FUNCTION_BLOCK Recipe_10017_DoubleCookiemitTopping
VAR_INPUT
	execute	: BOOL;
	Order	: DUT_RECIPEORDER;
END_VAR
VAR_OUTPUT
	RecipeInfo	: DUT_RECIPEOFFER;
	RecipeDone	: BOOL;	
	InitDone	: BOOL;
END_VAR
VAR
	StepDone	: BOOL;
	Layercnt	: INT := 0;
	OrderLayers	: INT := 1;
END_VAR

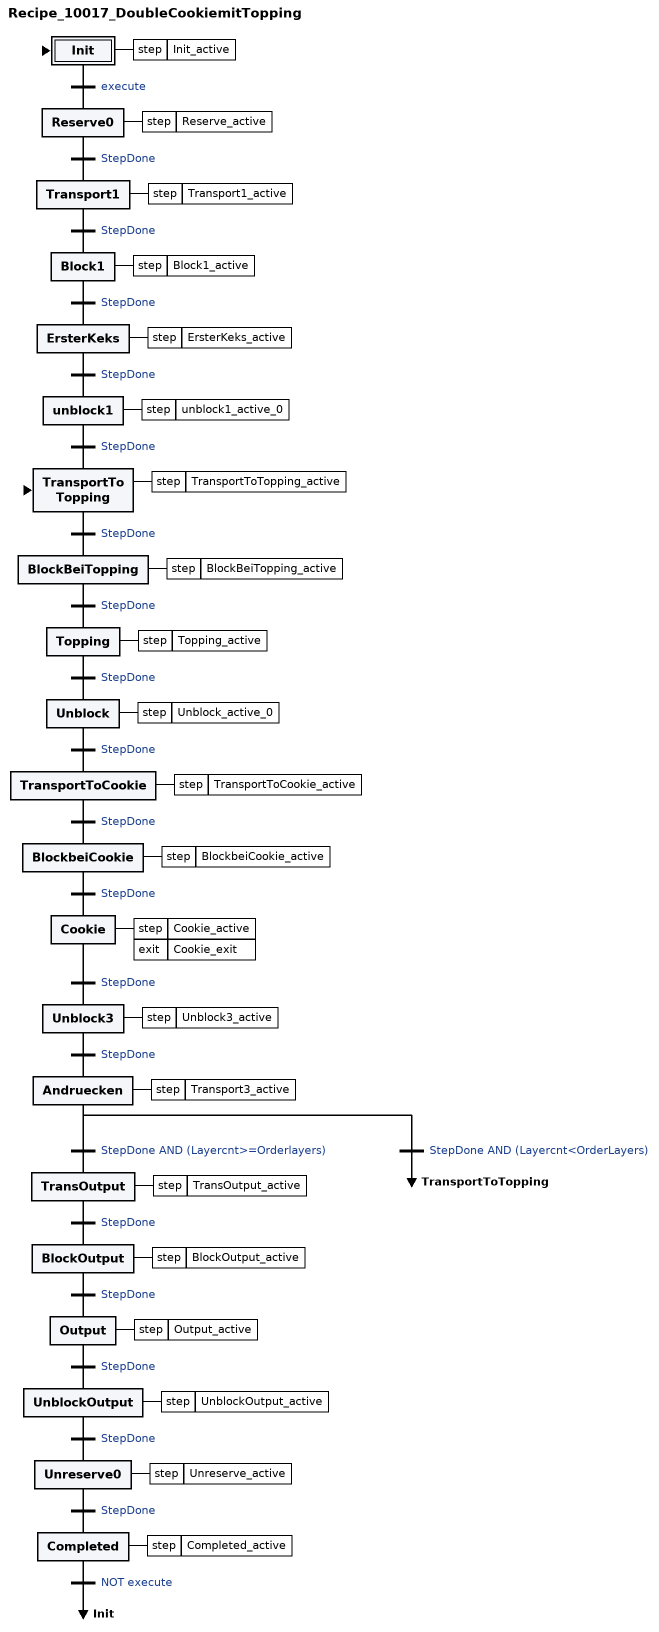
INITIAL_STEP Init:
    Init_active(N);  // step action
END_STEP
TRANSITION FROM Init TO Reserve0
    := execute;
END_TRANSITION
STEP Reserve0:
    Reserve_active(N);  // step action
END_STEP
TRANSITION FROM Reserve0 TO Transport1
    := StepDone;
END_TRANSITION
STEP Transport1:
    Transport1_active(N);  // step action
END_STEP
TRANSITION FROM Transport1 TO Block1
    := StepDone;
END_TRANSITION
STEP Block1:
    Block1_active(N);  // step action
END_STEP
TRANSITION FROM Block1 TO ErsterKeks
    := StepDone;
END_TRANSITION
STEP ErsterKeks:
    ErsterKeks_active(N);  // step action
END_STEP
TRANSITION FROM ErsterKeks TO unblock1
    := StepDone;
END_TRANSITION
STEP unblock1:
    unblock1_active_0(N);  // step action
END_STEP
TRANSITION FROM unblock1 TO TransportToTopping
    := StepDone;
END_TRANSITION
STEP TransportToTopping:
    TransportToTopping_active(N);  // step action
END_STEP
TRANSITION FROM TransportToTopping TO BlockBeiTopping
    := StepDone;
END_TRANSITION
STEP BlockBeiTopping:
    BlockBeiTopping_active(N);  // step action
END_STEP
TRANSITION FROM BlockBeiTopping TO Topping
    := StepDone;
END_TRANSITION
STEP Topping:
    Topping_active(N);  // step action
END_STEP
TRANSITION FROM Topping TO Unblock
    := StepDone;
END_TRANSITION
STEP Unblock:
    Unblock_active_0(N);  // step action
END_STEP
TRANSITION FROM Unblock TO TransportToCookie
    := StepDone;
END_TRANSITION
STEP TransportToCookie:
    TransportToCookie_active(N);  // step action
END_STEP
TRANSITION FROM TransportToCookie TO BlockbeiCookie
    := StepDone;
END_TRANSITION
STEP BlockbeiCookie:
    BlockbeiCookie_active(N);  // step action
END_STEP
TRANSITION FROM BlockbeiCookie TO Cookie
    := StepDone;
END_TRANSITION
STEP Cookie:
    Cookie_active(N);  // step action
    Cookie_exit(P0);  // exit action
END_STEP
TRANSITION FROM Cookie TO Unblock3
    := StepDone;
END_TRANSITION
STEP Unblock3:
    Unblock3_active(N);  // step action
END_STEP
TRANSITION FROM Unblock3 TO Andruecken
    := StepDone;
END_TRANSITION
STEP Andruecken:
    Transport3_active(N);  // step action
END_STEP
TRANSITION FROM Andruecken TO TransOutput
    := StepDone AND (Layercnt>=Orderlayers);
END_TRANSITION
STEP TransOutput:
    TransOutput_active(N);  // step action
END_STEP
TRANSITION FROM TransOutput TO BlockOutput
    := StepDone;
END_TRANSITION
STEP BlockOutput:
    BlockOutput_active(N);  // step action
END_STEP
TRANSITION FROM BlockOutput TO Output
    := StepDone;
END_TRANSITION
STEP Output:
    Output_active(N);  // step action
END_STEP
TRANSITION FROM Output TO UnblockOutput
    := StepDone;
END_TRANSITION
STEP UnblockOutput:
    UnblockOutput_active(N);  // step action
END_STEP
TRANSITION FROM UnblockOutput TO Unreserve0
    := StepDone;
END_TRANSITION
TRANSITION FROM Andruecken TO TransportToTopping
    := StepDone AND (Layercnt<OrderLayers);
END_TRANSITION
STEP Unreserve0:
    Unreserve_active(N);  // step action
END_STEP
TRANSITION FROM Unreserve0 TO Completed
    := StepDone;
END_TRANSITION
STEP Completed:
    Completed_active(N);  // step action
END_STEP
TRANSITION FROM Completed TO Init
    := NOT execute;
END_TRANSITION

ACTION unblock1_active_0:
StepDone := FALSE;

//Skill auswählen
ExecuteSkill.SkillID 		:= 1316;
ExecuteSkill.SkillName	 	:= 'Unblock';

//Parameter setzen

ExecuteSkill.Parameter[1].ID := 1;
ExecuteSkill.Parameter[1].Name := 'TaskID';
ExecuteSkill.Parameter[1].Value := 128 ;


(*
ExecuteSkill.Parameter[2].ID := ;
ExecuteSkill.Parameter[2].Name := '';
ExecuteSkill.Parameter[2].Value := ;
*)

(*
ExecuteSkill.Parameter[3].ID := ;
ExecuteSkill.Parameter[3].Name := '';
ExecuteSkill.Parameter[3].Value := ;
*)

(*
ExecuteSkill.Parameter[4].ID := ;
ExecuteSkill.Parameter[4].Name := '';
ExecuteSkill.Parameter[4].Value := ;
*)

(*
ExecuteSkill.Parameter[5].ID := ;
ExecuteSkill.Parameter[5].Name := '';
ExecuteSkill.Parameter[5].Value := ;
*)



ExecuteSkill();

StepDone := ExecuteSkill.Done;
END_ACTION

ACTION Topping_active:
StepDone := FALSE;

//Skill auswählen
CASE REAL_TO_INT (order.UserParameter[2*LayerCnt].Value) OF
	1: 
		ExecuteSkill.SkillID 		:=  1230;
		ExecuteSkill.SkillName	 	:= 'Strawberry Topping';
	2: 
		ExecuteSkill.SkillID 		:=  1240;
		ExecuteSkill.SkillName	 	:= 'Apple Topping';
	ELSE
		ExecuteSkill.SkillID 		:=  1230;
		ExecuteSkill.SkillName	 	:= 'Strawberry Topping';
END_CASE


//Parameter setzen

ExecuteSkill.Parameter[0].ID := 1;
ExecuteSkill.Parameter[0].Name := 'Amount';
ExecuteSkill.Parameter[0].Value := order.UserParameter[2*LayerCnt + 1].Value ;


(*
ExecuteSkill.Parameter[1].ID := 1;
ExecuteSkill.Parameter[1].Name := 'TaskID';
ExecuteSkill.Parameter[1].Value := 130;
*)
(*
ExecuteSkill.Parameter[2].ID := ;
ExecuteSkill.Parameter[2].Name := '';
ExecuteSkill.Parameter[2].Value := ;
*)

(*
ExecuteSkill.Parameter[3].ID := ;
ExecuteSkill.Parameter[3].Name := '';
ExecuteSkill.Parameter[3].Value := ;
*)

(*
ExecuteSkill.Parameter[4].ID := ;
ExecuteSkill.Parameter[4].Name := '';
ExecuteSkill.Parameter[4].Value := ;
*)

(*
ExecuteSkill.Parameter[5].ID := ;
ExecuteSkill.Parameter[5].Name := '';
ExecuteSkill.Parameter[5].Value := ;
*)

ExecuteSkill();

StepDone := ExecuteSkill.Done;
END_ACTION

ACTION Cookie_active:
StepDone := FALSE;
RecipeDone := FALSE;
//Skill auswählen
ExecuteSkill.SkillID 		:= 1010;
ExecuteSkill.SkillName	 	:= 'Cookie ausgeben';





ExecuteSkill();

StepDone := ExecuteSkill.Done;
END_ACTION

ACTION Transport3_active:
(*StepDone := FALSE;

//Skill auswählen
ExecuteSkill.SkillID 		:= 1320;
ExecuteSkill.SkillName	 	:= 'Transport';

//Parameter setzen

ExecuteSkill.Parameter[3].ID := 3;
ExecuteSkill.Parameter[3].Name := 'Velocity';
ExecuteSkill.Parameter[3].Value := 2800;



ExecuteSkill.Parameter[1].ID :=  1;
ExecuteSkill.Parameter[1].Name := 'TargetPosition X';
ExecuteSkill.Parameter[1].Value := 30 ;
ExecuteSkill.Parameter[1].StringValue := '#DP#-2#XPosition';



ExecuteSkill.Parameter[2].ID := 2;
ExecuteSkill.Parameter[2].Name := 'TargetPosition Z';
ExecuteSkill.Parameter[2].Value := 105;// ZCookieModule - ZCookieModuleCalibration - 2* Cookiethickness + toppingthickness+ Preasureheight  ;



ExecuteSkill.Parameter[4].ID := 4;
ExecuteSkill.Parameter[4].Name := 'Acceleration';
ExecuteSkill.Parameter[4].Value := 2000 ;


(*
ExecuteSkill.Parameter[5].ID := ;
ExecuteSkill.Parameter[5].Name := '';
ExecuteSkill.Parameter[5].Value := ;
*)



ExecuteSkill();

StepDone := ExecuteSkill.Done;
*)
StepDone := TRUE;
END_ACTION

ACTION Completed_active:
RecipeDone := TRUE;
StepDone := FALSE;
Layercnt := 0;
END_ACTION

ACTION BlockbeiCookie_active:
StepDone := FALSE;

//Skill auswählen
ExecuteSkill.SkillID 		:= 1315;
ExecuteSkill.SkillName	 	:= 'Block';

//Parameter setzen

ExecuteSkill.Parameter[1].ID := 1;
ExecuteSkill.Parameter[1].Name := 'TaskID';
ExecuteSkill.Parameter[1].Value := 130;


(*
ExecuteSkill.Parameter[2].ID := ;
ExecuteSkill.Parameter[2].Name := '';
ExecuteSkill.Parameter[2].Value := ;
*)

(*
ExecuteSkill.Parameter[3].ID := ;
ExecuteSkill.Parameter[3].Name := '';
ExecuteSkill.Parameter[3].Value := ;
*)

(*
ExecuteSkill.Parameter[4].ID := ;
ExecuteSkill.Parameter[4].Name := '';
ExecuteSkill.Parameter[4].Value := ;
*)

(*
ExecuteSkill.Parameter[5].ID := ;
ExecuteSkill.Parameter[5].Name := '';
ExecuteSkill.Parameter[5].Value := ;
*)



ExecuteSkill();

StepDone := ExecuteSkill.Done;
END_ACTION

ACTION BlockBeiTopping_active:
StepDone := FALSE;

//Skill auswählen
ExecuteSkill.SkillID 		:= 1315;
ExecuteSkill.SkillName	 	:= 'Block';

//Parameter setzen

ExecuteSkill.Parameter[1].ID := 1;
ExecuteSkill.Parameter[1].Name := 'TaskID';
ExecuteSkill.Parameter[1].Value := 130;


(*
ExecuteSkill.Parameter[2].ID := ;
ExecuteSkill.Parameter[2].Name := '';
ExecuteSkill.Parameter[2].Value := ;
*)

(*
ExecuteSkill.Parameter[3].ID := ;
ExecuteSkill.Parameter[3].Name := '';
ExecuteSkill.Parameter[3].Value := ;
*)

(*
ExecuteSkill.Parameter[4].ID := ;
ExecuteSkill.Parameter[4].Name := '';
ExecuteSkill.Parameter[4].Value := ;
*)

(*
ExecuteSkill.Parameter[5].ID := ;
ExecuteSkill.Parameter[5].Name := '';
ExecuteSkill.Parameter[5].Value := ;
*)



ExecuteSkill();

StepDone := ExecuteSkill.Done;
END_ACTION

ACTION ErsterKeks_active:
StepDone := FALSE;
RecipeDone := FALSE;
//Skill auswählen
ExecuteSkill.SkillID 		:= 1010;
ExecuteSkill.SkillName	 	:= 'Seperate Cookie';


ExecuteSkill();

StepDone := ExecuteSkill.Done;
END_ACTION

ACTION Transport1_active:
StepDone := FALSE;

//Skill auswählen
ExecuteSkill.SkillID 		:= 1320;
ExecuteSkill.SkillName	 	:= 'Transport';

//Parameter setzen

ExecuteSkill.Parameter[3].ID := 3;
ExecuteSkill.Parameter[3].Name := 'Velocity';
ExecuteSkill.Parameter[3].Value := 1500;



ExecuteSkill.Parameter[4].ID := 4 ;
ExecuteSkill.Parameter[4].Name := 'Acceleration';
ExecuteSkill.Parameter[4].Value := 1000 ;



ExecuteSkill.Parameter[1].ID := 1;
ExecuteSkill.Parameter[1].Name := 'TargetPosition X';
ExecuteSkill.Parameter[1].Value := 3200 ;
ExecuteSkill.Parameter[1].StringValue := '#DP#2#XPosition' ;




ExecuteSkill.Parameter[2].ID := 2;
ExecuteSkill.Parameter[2].Name := 'TargetPosition Z';
ExecuteSkill.Parameter[2].Value := ZCookieModule + ZCocktailModuleCalibration;


(*
ExecuteSkill.Parameter[5].ID := ;
ExecuteSkill.Parameter[5].Name := '';
ExecuteSkill.Parameter[5].Value := ;
*)



ExecuteSkill();

StepDone := ExecuteSkill.Done;
END_ACTION

ACTION Production0_active:
StepDone := FALSE;
RecipeDone := FALSE; 
//simulation ausgewählt?
CASE LREAL_TO_INT (order.UserParameter[2].Value) OF

1:
ExecuteSkill.SkillID 		:= 1337;
ExecuteSkill.SkillName	 	:= 'Testskill';

ExecuteSkill();

StepDone := ExecuteSkill.Done;
ELSE StepDone := TRUE;

END_CASE
END_ACTION

ACTION TransportToTopping_active:
StepDone := FALSE;

//Skill auswählen
ExecuteSkill.SkillID 		:= 1320;
ExecuteSkill.SkillName	 	:= 'Transport';

//Parameter setzen

ExecuteSkill.Parameter[3].ID := 3;
ExecuteSkill.Parameter[3].Name := 'Velocity';
ExecuteSkill.Parameter[3].Value := 1000;



ExecuteSkill.Parameter[1].ID :=  1;
ExecuteSkill.Parameter[1].Name := 'TargetPosition X';
ExecuteSkill.Parameter[1].Value := 30 ;
ExecuteSkill.Parameter[1].StringValue := '#DP#2#XPosition';



ExecuteSkill.Parameter[2].ID := 2;
ExecuteSkill.Parameter[2].Name := 'TargetPosition Z';
ExecuteSkill.Parameter[2].Value := ZCremeModule + ZCremeModuleCalibration - Layercnt * ( cookiethickness + toppingthickness);

ExecuteSkill();

StepDone := ExecuteSkill.Done;
END_ACTION

ACTION UnblockOutput_active:
StepDone := FALSE;

//Skill auswählen
ExecuteSkill.SkillID 		:= 1316;
ExecuteSkill.SkillName	 	:= 'Unblock';

//Parameter setzen



(*
ExecuteSkill.Parameter[2].ID := ;
ExecuteSkill.Parameter[2].Name := '';
ExecuteSkill.Parameter[2].Value := ;
*)

(*
ExecuteSkill.Parameter[3].ID := ;
ExecuteSkill.Parameter[3].Name := '';
ExecuteSkill.Parameter[3].Value := ;
*)

(*
ExecuteSkill.Parameter[4].ID := ;
ExecuteSkill.Parameter[4].Name := '';
ExecuteSkill.Parameter[4].Value := ;
*)

(*
ExecuteSkill.Parameter[5].ID := ;
ExecuteSkill.Parameter[5].Name := '';
ExecuteSkill.Parameter[5].Value := ;
*)



ExecuteSkill();

StepDone := ExecuteSkill.Done;
END_ACTION

ACTION BlockOutput_active:
StepDone := FALSE;

//Skill auswählen



ExecuteSkill.SkillID 		:= 1315;
ExecuteSkill.SkillName	 	:= 'Block';

ExecuteSkill();

StepDone := ExecuteSkill.Done;
END_ACTION

ACTION Transport_active:
StepDone := FALSE;

//Skill auswählen

CASE LREAL_TO_INT (order.UserParameter[2].Value) OF

1:
//Skill auswählen
ExecuteSkill.SkillID 		:= 1320;
ExecuteSkill.SkillName	 	:= 'Transport';

//Parameter setzen

ExecuteSkill.Parameter[3].ID :=3 ;
ExecuteSkill.Parameter[3].Name := 'Velocity';
ExecuteSkill.Parameter[3].Value := 1500;



ExecuteSkill.Parameter[1].ID :=1 ;
ExecuteSkill.Parameter[1].Name := 'TargetPosition X';
ExecuteSkill.Parameter[1].StringValue := '#DP#2#XPosition';
ExecuteSkill.Parameter[1].Value := 200 ;


ExecuteSkill.Parameter[2].ID := 2 ;
ExecuteSkill.Parameter[2].Name := 'TargetPosition Z';
ExecuteSkill.Parameter[2].Value := 90 ;



ExecuteSkill.Parameter[4].ID := 4 ;
ExecuteSkill.Parameter[4].Name := 'Acceleration';
ExecuteSkill.Parameter[4].Value := 4500;


(*
ExecuteSkill.Parameter[5].ID := ;
ExecuteSkill.Parameter[5].Name := '';
ExecuteSkill.Parameter[5].Value := ;
*)



ExecuteSkill();

StepDone := ExecuteSkill.Done;
ELSE StepDone := TRUE;

END_CASE
END_ACTION

ACTION Unblock_active:
StepDone := FALSE;

//Skill auswählen
ExecuteSkill.SkillID 		:= 1316;
ExecuteSkill.SkillName	 	:= 'Unblock';

//Parameter setzen

ExecuteSkill.Parameter[1].ID := 1;
ExecuteSkill.Parameter[1].Name := 'TaskID';
ExecuteSkill.Parameter[1].Value := 125;


(*
ExecuteSkill.Parameter[2].ID := ;
ExecuteSkill.Parameter[2].Name := '';
ExecuteSkill.Parameter[2].Value := ;
*)

(*
ExecuteSkill.Parameter[3].ID := ;
ExecuteSkill.Parameter[3].Name := '';
ExecuteSkill.Parameter[3].Value := ;
*)

(*
ExecuteSkill.Parameter[4].ID := ;
ExecuteSkill.Parameter[4].Name := '';
ExecuteSkill.Parameter[4].Value := ;
*)

(*
ExecuteSkill.Parameter[5].ID := ;
ExecuteSkill.Parameter[5].Name := '';
ExecuteSkill.Parameter[5].Value := ;
*)



ExecuteSkill();

StepDone := ExecuteSkill.Done;
END_ACTION

ACTION Production2_active:
StepDone := FALSE;
RecipeDone := FALSE;
//Skill auswählen
ExecuteSkill.SkillID 		:= 1339;
ExecuteSkill.SkillName	 	:= 'ParameterTESTSKILL1339';


ExecuteSkill.Parameter[0].ID := 10;
ExecuteSkill.Parameter[0].Name := 'Blinkfrequenz';
ExecuteSkill.Parameter[0].Value := Order.UserParameter[0].Value*2;


ExecuteSkill();

StepDone := ExecuteSkill.Done;
END_ACTION

ACTION Unblock3_active:
StepDone := FALSE;

//Skill auswählen
ExecuteSkill.SkillID 		:= 1316;
ExecuteSkill.SkillName	 	:= 'Unblock';

//Parameter setzen

ExecuteSkill.Parameter[1].ID := 1;
ExecuteSkill.Parameter[1].Name := 'TaskID';
ExecuteSkill.Parameter[1].Value := 131;


(*
ExecuteSkill.Parameter[2].ID := ;
ExecuteSkill.Parameter[2].Name := '';
ExecuteSkill.Parameter[2].Value := ;
*)

(*
ExecuteSkill.Parameter[3].ID := ;
ExecuteSkill.Parameter[3].Name := '';
ExecuteSkill.Parameter[3].Value := ;
*)

(*
ExecuteSkill.Parameter[4].ID := ;
ExecuteSkill.Parameter[4].Name := '';
ExecuteSkill.Parameter[4].Value := ;
*)

(*
ExecuteSkill.Parameter[5].ID := ;
ExecuteSkill.Parameter[5].Name := '';
ExecuteSkill.Parameter[5].Value := ;
*)



ExecuteSkill();

StepDone := ExecuteSkill.Done;
END_ACTION

ACTION ST40_TransOutput_active:
//RT: 2014.11.23: Mover zum Output
StepDone := FALSE;

//Skill auswählen
ExecuteSkill.SkillID 		:= 1320;
ExecuteSkill.SkillName	 	:= 'Transport';

//Parameter setzen

ExecuteSkill.Parameter[3].ID := 3;
ExecuteSkill.Parameter[3].Name := 'Velocity';
ExecuteSkill.Parameter[3].Value := 300;



ExecuteSkill.Parameter[1].ID :=  1;
ExecuteSkill.Parameter[1].Name := 'TargetPosition X';
ExecuteSkill.Parameter[1].Value := 30 ;
ExecuteSkill.Parameter[1].StringValue := '#DP#2#XPosition';



ExecuteSkill.Parameter[2].ID := 2;
ExecuteSkill.Parameter[2].Name := 'TargetPosition Z';
ExecuteSkill.Parameter[2].Value := ZInputOutput;// ZCookieModule - ZCookieModuleCalibration - 2* Cookiethickness + toppingthickness+ Preasureheight  ;



(* ExecuteSkill.Parameter[4].ID := 4;
ExecuteSkill.Parameter[4].Name := 'Acceleration';
ExecuteSkill.Parameter[4].Value :=0 ;

*)
(*
ExecuteSkill.Parameter[5].ID := ;
ExecuteSkill.Parameter[5].Name := '';
ExecuteSkill.Parameter[5].Value := ;
*)



ExecuteSkill();

StepDone := ExecuteSkill.Done;
END_ACTION

ACTION Block2_active:
StepDone := FALSE;

//Skill auswählen
ExecuteSkill.SkillID 		:= 1315;
ExecuteSkill.SkillName	 	:= 'Block';

//Parameter setzen

ExecuteSkill.Parameter[1].ID := 1;
ExecuteSkill.Parameter[1].Name := 'TaskID';
ExecuteSkill.Parameter[1].Value := 130;


(*
ExecuteSkill.Parameter[2].ID := ;
ExecuteSkill.Parameter[2].Name := '';
ExecuteSkill.Parameter[2].Value := ;
*)

(*
ExecuteSkill.Parameter[3].ID := ;
ExecuteSkill.Parameter[3].Name := '';
ExecuteSkill.Parameter[3].Value := ;
*)

(*
ExecuteSkill.Parameter[4].ID := ;
ExecuteSkill.Parameter[4].Name := '';
ExecuteSkill.Parameter[4].Value := ;
*)

(*
ExecuteSkill.Parameter[5].ID := ;
ExecuteSkill.Parameter[5].Name := '';
ExecuteSkill.Parameter[5].Value := ;
*)



ExecuteSkill();

StepDone := ExecuteSkill.Done;
END_ACTION

ACTION Unblock2_active:
StepDone := FALSE;

//Skill auswählen
ExecuteSkill.SkillID 		:= 1316;
ExecuteSkill.SkillName	 	:= 'Unblock';

//Parameter setzen

ExecuteSkill.Parameter[1].ID := 1;
ExecuteSkill.Parameter[1].Name := 'TaskID';
ExecuteSkill.Parameter[1].Value := 131;


(*
ExecuteSkill.Parameter[2].ID := ;
ExecuteSkill.Parameter[2].Name := '';
ExecuteSkill.Parameter[2].Value := ;
*)

(*
ExecuteSkill.Parameter[3].ID := ;
ExecuteSkill.Parameter[3].Name := '';
ExecuteSkill.Parameter[3].Value := ;
*)

(*
ExecuteSkill.Parameter[4].ID := ;
ExecuteSkill.Parameter[4].Name := '';
ExecuteSkill.Parameter[4].Value := ;
*)

(*
ExecuteSkill.Parameter[5].ID := ;
ExecuteSkill.Parameter[5].Name := '';
ExecuteSkill.Parameter[5].Value := ;
*)



ExecuteSkill();

StepDone := ExecuteSkill.Done;
END_ACTION

ACTION TransOutput_active:
StepDone := FALSE;

//Skill auswählen
ExecuteSkill.SkillID 		:= 1320;
ExecuteSkill.SkillName	 	:= 'Transport';

//Parameter setzen

ExecuteSkill.Parameter[3].ID := 3;
ExecuteSkill.Parameter[3].Name := 'Velocity';
ExecuteSkill.Parameter[3].Value := 280;



ExecuteSkill.Parameter[1].ID :=  1;
ExecuteSkill.Parameter[1].Name := 'TargetPosition X';
ExecuteSkill.Parameter[1].Value := 30 ;
ExecuteSkill.Parameter[1].StringValue := '#DP#2#XPosition';



ExecuteSkill.Parameter[2].ID := 2;
ExecuteSkill.Parameter[2].Name := 'TargetPosition Z';
ExecuteSkill.Parameter[2].Value := ZInputOutput;// ZCookieModule - ZCookieModuleCalibration - 2* Cookiethickness + toppingthickness+ Preasureheight  ;



(* ExecuteSkill.Parameter[4].ID := 4;
ExecuteSkill.Parameter[4].Name := 'Acceleration';
ExecuteSkill.Parameter[4].Value :=0 ;

*)
(*
ExecuteSkill.Parameter[5].ID := ;
ExecuteSkill.Parameter[5].Name := '';
ExecuteSkill.Parameter[5].Value := ;
*)



ExecuteSkill();

StepDone := ExecuteSkill.Done;
END_ACTION

ACTION Cookie_exit:
Layercnt := Layercnt +1;
END_ACTION

ACTION Unblock1_active:
StepDone := FALSE;

//Skill auswählen

CASE LREAL_TO_INT (order.UserParameter[2].Value) OF

1:
ExecuteSkill.SkillID 		:= 1316;
ExecuteSkill.SkillName	 	:= 'Unblock';

ExecuteSkill();

StepDone := ExecuteSkill.Done;
ELSE StepDone := TRUE;

END_CASE
END_ACTION

ACTION Output_active:
StepDone := FALSE;

//Skill auswählen
ExecuteSkill.SkillID 		:= 1403;
ExecuteSkill.SkillName	 	:= 'Output';

//Parameter setzen

ExecuteSkill.Parameter[1].ID := 1;
ExecuteSkill.Parameter[1].Name := 'TaskID';
ExecuteSkill.Parameter[1].Value := Order.TaskID;


(*
ExecuteSkill.Parameter[2].ID := ;
ExecuteSkill.Parameter[2].Name := '';
ExecuteSkill.Parameter[2].Value := ;
*)

(*
ExecuteSkill.Parameter[3].ID := ;
ExecuteSkill.Parameter[3].Name := '';
ExecuteSkill.Parameter[3].Value := ;
*)

(*
ExecuteSkill.Parameter[4].ID := ;
ExecuteSkill.Parameter[4].Name := '';
ExecuteSkill.Parameter[4].Value := ;
*)

(*
ExecuteSkill.Parameter[5].ID := ;
ExecuteSkill.Parameter[5].Name := '';
ExecuteSkill.Parameter[5].Value := ;
*)



ExecuteSkill();

StepDone := ExecuteSkill.Done;
END_ACTION

ACTION Block1_active:
StepDone := FALSE;

//Skill auswählen
ExecuteSkill.SkillID 		:= 1315;
ExecuteSkill.SkillName	 	:= 'Block';

//Parameter setzen

ExecuteSkill.Parameter[1].ID := 1;
ExecuteSkill.Parameter[1].Name := 'TaskID';
ExecuteSkill.Parameter[1].Value := 127;


(*
ExecuteSkill.Parameter[2].ID := ;
ExecuteSkill.Parameter[2].Name := '';
ExecuteSkill.Parameter[2].Value := ;
*)

(*
ExecuteSkill.Parameter[3].ID := ;
ExecuteSkill.Parameter[3].Name := '';
ExecuteSkill.Parameter[3].Value := ;
*)

(*
ExecuteSkill.Parameter[4].ID := ;
ExecuteSkill.Parameter[4].Name := '';
ExecuteSkill.Parameter[4].Value := ;
*)

(*
ExecuteSkill.Parameter[5].ID := ;
ExecuteSkill.Parameter[5].Name := '';
ExecuteSkill.Parameter[5].Value := ;
*)



ExecuteSkill();

StepDone := ExecuteSkill.Done;
END_ACTION

ACTION Block0_active:
StepDone := FALSE;

//Skill auswählen

CASE LREAL_TO_INT (order.UserParameter[2].Value) OF

1:
ExecuteSkill.SkillID 		:= 1315;
ExecuteSkill.SkillName	 	:= 'Block';

ExecuteSkill();

StepDone := ExecuteSkill.Done;
ELSE StepDone := TRUE;

END_CASE
END_ACTION

ACTION Unreserve_active:
StepDone := FALSE;

//Skill auswählen
ExecuteSkill.SkillID 		:= 1311;
ExecuteSkill.SkillName	 	:= 'Unreserve';

//Parameter setzen

ExecuteSkill.Parameter[1].ID := 1;
ExecuteSkill.Parameter[1].Name := 'TaskID';
ExecuteSkill.Parameter[1].Value := 131;


(*
ExecuteSkill.Parameter[2].ID := ;
ExecuteSkill.Parameter[2].Name := '';
ExecuteSkill.Parameter[2].Value := ;
*)

(*
ExecuteSkill.Parameter[3].ID := ;
ExecuteSkill.Parameter[3].Name := '';
ExecuteSkill.Parameter[3].Value := ;
*)

(*
ExecuteSkill.Parameter[4].ID := ;
ExecuteSkill.Parameter[4].Name := '';
ExecuteSkill.Parameter[4].Value := ;
*)

(*
ExecuteSkill.Parameter[5].ID := ;
ExecuteSkill.Parameter[5].Name := '';
ExecuteSkill.Parameter[5].Value := ;
*)



ExecuteSkill();

StepDone := ExecuteSkill.Done;
END_ACTION

ACTION Init_active:
RecipeDone := FALSE;

// Initialisation of Recipe Parameters an name etc
RecipeInfo.Name := 'Double Cookie';
RecipeInfo.Description := 'Butter Cookies framing your choosen Topping';
RecipeInfo.Dummy := FALSE;
RecipeInfo.RecipeID := 10017;	// 
Initdone := TRUE;


//Parameter 0:

	RecipeInfo.UserParameter[0].Dummy 		:= FALSE;
	RecipeInfo.UserParameter[0].Default		:= 1;
	RecipeInfo.UserParameter[0].Description	:= 'Choose your first Topping (Top Layer)';
	RecipeInfo.UserParameter[0].MaxValue	:= 2;
	RecipeInfo.UserParameter[0].MinValue	:= 1;
	RecipeInfo.UserParameter[0].Name		:= 'Topping';
	RecipeInfo.UserParameter[0].Unit		:= 'Strawberry, Apple';
	RecipeInfo.UserParameter[0].Step		:= 1;

//Parameter 1:

	RecipeInfo.UserParameter[1].Dummy 		:= FALSE;
	RecipeInfo.UserParameter[1].Default		:= 50;
	RecipeInfo.UserParameter[1].Description	:= 'Amount of the selected Topping';
	RecipeInfo.UserParameter[1].MaxValue	:= 100;
	RecipeInfo.UserParameter[1].MinValue	:= 0;
	RecipeInfo.UserParameter[1].Name		:= 'Amount';
	RecipeInfo.UserParameter[1].Unit		:= '';
	RecipeInfo.UserParameter[1].Step		:= 1;

//Parameter 2:
	(*RecipeInfo.UserParameter[2].Dummy 		:= FALSE;
	RecipeInfo.UserParameter[2].Default		:= 2;
	RecipeInfo.UserParameter[2].Description	:= 'Choose weather you want to include a simulated module';
	RecipeInfo.UserParameter[2].MaxValue	:= 2;
	RecipeInfo.UserParameter[2].MinValue	:= 1;
	RecipeInfo.UserParameter[2].Name		:= 'Virtual Module';
	RecipeInfo.UserParameter[2].Unit		:= 'enabled, disabled';
	RecipeInfo.UserParameter[2].Step		:= 1;*)
(*
//Parameter 3:
	RecipeInfo.UserParameter[3].Dummy 		:= FALSE;
	RecipeInfo.UserParameter[3].Default		:= 1;
	RecipeInfo.UserParameter[3].Description	:= 'Amount of the selected Topping';
	RecipeInfo.UserParameter[3].MaxValue	:= 100;
	RecipeInfo.UserParameter[3].MinValue	:= 0;
	RecipeInfo.UserParameter[3].Name		:= 'Amount';
	RecipeInfo.UserParameter[3].Unit		:= '';
	RecipeInfo.UserParameter[3].Step		:= 1;
//Parameter 4:

	RecipeInfo.UserParameter[4].Dummy 		:= FALSE;
	RecipeInfo.UserParameter[4].Default		:= 1;
	RecipeInfo.UserParameter[4].Description	:= 'Choose your third Topping';
	RecipeInfo.UserParameter[4].MaxValue	:= 2;
	RecipeInfo.UserParameter[4].MinValue	:= 1;
	RecipeInfo.UserParameter[4].Name		:= 'Topping';
	RecipeInfo.UserParameter[4].Unit		:= 'Strawberry, Apple';
	RecipeInfo.UserParameter[4].Step		:= 1;
//Parameter 5:

	RecipeInfo.UserParameter[5].Dummy 		:= FALSE;
	RecipeInfo.UserParameter[5].Default		:= 50;
	RecipeInfo.UserParameter[5].Description	:= 'Amount of the selected Topping';
	RecipeInfo.UserParameter[5].MaxValue	:= 100;
	RecipeInfo.UserParameter[5].MinValue	:= 0;
	RecipeInfo.UserParameter[5].Name		:= 'Amount';
	RecipeInfo.UserParameter[5].Unit		:= '';
	RecipeInfo.UserParameter[5].Step		:= 1;
*)
END_ACTION

ACTION TransportToCookie_active:
StepDone := FALSE;

//Skill auswählen
ExecuteSkill.SkillID 		:= 1320;
ExecuteSkill.SkillName	 	:= 'Transport';

//Parameter setzen

ExecuteSkill.Parameter[3].ID := 3;
ExecuteSkill.Parameter[3].Name := 'Velocity';
ExecuteSkill.Parameter[3].Value := 400;



ExecuteSkill.Parameter[1].ID :=  1;
ExecuteSkill.Parameter[1].Name := 'TargetPosition X';
ExecuteSkill.Parameter[1].Value := 30 ;
ExecuteSkill.Parameter[1].StringValue := '#DP#2#XPosition';



ExecuteSkill.Parameter[2].ID := 2;
ExecuteSkill.Parameter[2].Name := 'TargetPosition Z';
ExecuteSkill.Parameter[2].Value := ZCookieModule + ZCookieModuleCalibration - ((Layercnt +1) * ( toppingthickness + cookiethickness)) ;

ExecuteSkill();

StepDone := ExecuteSkill.Done;
END_ACTION

ACTION Reserve_active:
StepDone := FALSE;
RecipeDone := FALSE;
//Skill auswählen
ExecuteSkill.SkillID 		:= 1310;
ExecuteSkill.SkillName	 	:= 'Reserve';

//Parameter setzen

ExecuteSkill.Parameter[1].ID := 1;
ExecuteSkill.Parameter[1].Name := 'TaskID';
ExecuteSkill.Parameter[1].Value := 123;


(*
ExecuteSkill.Parameter[2].ID := ;
ExecuteSkill.Parameter[2].Name := '';
ExecuteSkill.Parameter[2].Value := ;
*)

(*
ExecuteSkill.Parameter[3].ID := ;
ExecuteSkill.Parameter[3].Name := '';
ExecuteSkill.Parameter[3].Value := ;
*)

(*
ExecuteSkill.Parameter[4].ID := ;
ExecuteSkill.Parameter[4].Name := '';
ExecuteSkill.Parameter[4].Value := ;
*)

(*
ExecuteSkill.Parameter[5].ID := ;
ExecuteSkill.Parameter[5].Name := '';
ExecuteSkill.Parameter[5].Value := ;
*)



ExecuteSkill();

StepDone := ExecuteSkill.Done;
END_ACTION

ACTION Unblock_active_0:
StepDone := FALSE;

//Skill auswählen
ExecuteSkill.SkillID 		:= 1316;
ExecuteSkill.SkillName	 	:= 'Unblock';

//Parameter setzen

ExecuteSkill.Parameter[1].ID := 1;
ExecuteSkill.Parameter[1].Name := 'TaskID';
ExecuteSkill.Parameter[1].Value := 128 ;


(*
ExecuteSkill.Parameter[2].ID := ;
ExecuteSkill.Parameter[2].Name := '';
ExecuteSkill.Parameter[2].Value := ;
*)

(*
ExecuteSkill.Parameter[3].ID := ;
ExecuteSkill.Parameter[3].Name := '';
ExecuteSkill.Parameter[3].Value := ;
*)

(*
ExecuteSkill.Parameter[4].ID := ;
ExecuteSkill.Parameter[4].Name := '';
ExecuteSkill.Parameter[4].Value := ;
*)

(*
ExecuteSkill.Parameter[5].ID := ;
ExecuteSkill.Parameter[5].Name := '';
ExecuteSkill.Parameter[5].Value := ;
*)



ExecuteSkill();

StepDone := ExecuteSkill.Done;
END_ACTION

ACTION Transport2_active:
StepDone := FALSE;

//Skill auswählen
ExecuteSkill.SkillID 		:= 1320;
ExecuteSkill.SkillName	 	:= 'Transport';

//Parameter setzen

ExecuteSkill.Parameter[3].ID := 3;
ExecuteSkill.Parameter[3].Name := 'Velocity';
ExecuteSkill.Parameter[3].Value := 2800;



ExecuteSkill.Parameter[1].ID :=  1;
ExecuteSkill.Parameter[1].Name := 'TargetPosition X';
ExecuteSkill.Parameter[1].Value := 30 ;
ExecuteSkill.Parameter[1].StringValue := '#DP#2#XPosition';



ExecuteSkill.Parameter[2].ID := 2;
ExecuteSkill.Parameter[2].Name := 'TargetPosition Z';
ExecuteSkill.Parameter[2].Value := 0 ;



ExecuteSkill.Parameter[4].ID := 4;
ExecuteSkill.Parameter[4].Name := 'Acceleration';
ExecuteSkill.Parameter[4].Value := 2000 ;


(*
ExecuteSkill.Parameter[5].ID := ;
ExecuteSkill.Parameter[5].Name := '';
ExecuteSkill.Parameter[5].Value := ;
*)



ExecuteSkill();

StepDone := ExecuteSkill.Done;
END_ACTION

END_FUNCTION_BLOCK

(* stored: Version 1.1.0.1, ProductVersion 3.1.0.25
   POU Recipe_10017_DoubleCookiemitTopping: Id {e9291349-8e41-4208-9582-332a7729ee8f}
   Action unblock1_active_0: Id {063a34a4-c2ac-4806-b2ec-d7226a64a59a}
   Action Topping_active: Id {09be58b5-d02d-44ce-8bb7-3a0cc7fe133c}
   Action Cookie_active: Id {0ae03135-3cd8-45e5-aa05-32b804ff7d32}
   Action Transport3_active: Id {198b2c43-dcd3-4122-bfa3-00e0a8a25f35}
   Action Completed_active: Id {22632304-23eb-42cf-85d8-f7e733018428}
   Action BlockbeiCookie_active: Id {238f9ae3-f226-4eea-9366-332133a24033}
   Action BlockBeiTopping_active: Id {26795436-a644-472f-b717-cf72548e18d3}
   Action ErsterKeks_active: Id {28fc033c-7e90-4310-ac82-42d5dda9b278}
   Action Transport1_active: Id {3217c8d7-21e7-4458-bf40-b3f940b3f36e}
   Action Production0_active: Id {32d794f6-c01e-407c-99d2-7b1435c2a0c2}
   Action TransportToTopping_active: Id {362f5d4c-0c22-46b9-9307-955098d3dbb3}
   Action UnblockOutput_active: Id {4bfafa66-44d9-40ca-9d3f-aecf15070060}
   Action BlockOutput_active: Id {4e9ed973-62ff-4898-adf6-8371fffc81b4}
   Action Transport_active: Id {6770f680-6a56-45e1-a6c0-8bb978c9fa1c}
   Action Unblock_active: Id {888ab9db-c8cc-42ab-9d43-97b0773ce4c9}
   Action Production2_active: Id {8c101efb-d2f6-4a19-85bf-eb5cd180d657}
   Action Unblock3_active: Id {95a2d72f-18b8-48ac-8083-1f205155f339}
   Action ST40_TransOutput_active: Id {9d0a2509-2a81-4cf2-bde0-368e2f2bbc11}
   Action Block2_active: Id {a36a84f5-740e-453d-8b17-dc98ba9b9a7a}
   Action Unblock2_active: Id {a95c4a78-cfa0-4b48-b059-9a1ee40f2edd}
   Action TransOutput_active: Id {b1b65a99-44a8-4dcb-99c9-81bdc02ceccf}
   Action Cookie_exit: Id {b7dcb812-4bfc-40d4-92e4-2e7743162fe0}
   Action Unblock1_active: Id {b87d9d90-ef7c-4277-894e-873c5d9a8c7a}
   Action Output_active: Id {ba7d08a9-eba8-4ab1-ae13-b964969af111}
   Action Block1_active: Id {c05976ca-e386-4de7-a7a8-d0036cc38e0c}
   Action Block0_active: Id {c9765f3a-6c8d-47c5-8de9-c710eb471848}
   Action Unreserve_active: Id {cd08b063-e5e6-4b31-88b6-930387e79248}
   Action Init_active: Id {cf29ca48-b739-48cc-933c-d45543afbadf}
   Action TransportToCookie_active: Id {e0dcd238-3faf-4537-9d70-a5905e8f039c}
   Action Reserve_active: Id {e9f18f40-9a2e-4a07-90ee-c151a398dd40}
   Action Unblock_active_0: Id {f5a6224a-de7f-47ce-b6da-e2f4d6898d96}
   Action Transport2_active: Id {f68d8fb6-1baf-45c4-aeae-b99b38474b95} *)
